(* PLC project conveyor1, Dassault Systèmes ControlBuild 2024x *)
(* stored: creationDateTime 2023-10-03T11:13:53-01:00 *)

FUNCTION_BLOCK tri_chain.conveyor1
  VAR_INPUT
    linearSpeed : REAL := 0.0;
  END_VAR
  VAR
    status_act_prod : DINT := 0;
    m11 : REAL := 1.0;
    m12 : REAL := 0.0;
    m13 : REAL := 0.0;
    m14 : REAL := 0.0;
    m21 : REAL := 0.0;
    m22 : REAL := 1.0;
    m23 : REAL := 0.0;
    m24 : REAL := 0.0;
    m31 : REAL := 0.0;
    m32 : REAL := 0.0;
    m33 : REAL := 1.0;
    m34 : REAL := 0.0;
    m41 : REAL := 0.0;
    m42 : REAL := 0.0;
    m43 : REAL := 0.0;
    m44 : REAL := 1.0;
    px : REAL := 0.0;
    py : REAL := 0.0;
    pz : REAL := 0.0;
    dx : REAL := 0.0;
    dy : REAL := 0.0;
    dz : REAL := 0.0;
    sProduct : REAL := 0.0;
    interaction : BOOL := false;
  END_VAR
  VAR
    d_locking : BOOL := false;
    v_d_locking : BOOL := false;
  END_VAR


ACTION C_source_code:
/* ----------------------------------------------------------------	*/
/* Type : Model of Operative Behaviour					*/
/* Category :  Conveyor							*/
/* Author : Dassault Systemes						*/
/* Update date : June 2018							*/
/* ----------------------------------------------------------------	*/

/* -----------------------------------------------------------------	*/
/* px, py et pz are the lowest coordinates.				*/
/* dx, dy et dz are the actor's dimensions 				*/
/* sProduct is the absolute speed given to the product.		*/
/*	CLOCK_PERIOD returns the cycle time in 1000th. of ms		*/
/* The linear speed is given in mm/s.					*/
/* -----------------------------------------------------------------	*/

if (!d_locking)
	{
	sProduct=linearSpeed*(CLOCK_PERIOD/1000000);
	}
else sProduct=0;
END_ACTION
END_FUNCTION_BLOCK
